// Controls the heater
//
FUNCTION_BLOCK FB_HeaterCtrl
VAR_INPUT
	
	Step: SINT; // Step counter (1...100)
	
END_VAR
VAR
	
	// Function blocks...
	fbPID: FB_CTRL_PID; // PID controller
	
	// Structures...
	stParams: ST_CTRL_PID_PARAMS; // PID controller parameters
	
	// Booleans...
	bInitialized: BOOL; // Initialized
	bRestart:     BOOL; // Restart
	bAutoStep:    BOOL; // Auto-step
	
END_VAR

// Initialize members
bRestart    := ( bRestart    OR IO_Outputs.o_Restart );

// First visit ? 
IF NOT bInitialized THEN
	
	// Initialize PID controller parameters
	bInitialized := TRUE;
	InitPidParams( ADR( stParams ));
	
	bAutoStep := FALSE;
	
END_IF

// Is the the starting step ?
IF Step = 1 THEN
  
	// Update the PID controller once per every second
	fbPID
	(
		fSetpointValue := gSetpoint,
		fActualValue   := IO_Inputs.i_HtrTemp,
		fManSyncValue  := 0,
		bSync          := FALSE,
		eMode          := SEL( bRestart, eCTRL_MODE_ACTIVE, eCTRL_MODE_RESET ),
		bHold          := FALSE,
		stParams       := stParams,
		fOut           => gPower,
		eState         => gePidState
(*
		bARWactive     => BOOL;
		eErrorId       => E_CTRL_ERRORCODES;
		bError         => BOOL;
*)
	);

	// Control the heater to ON/OFF
	IO_Outputs.o_HtrON := ( fbPID.fOut >= Step );
	bRestart           := FALSE;
	
	// Auto-step control
	IF bAutoStep THEN
		gAutoStepTimer := gAutoStepTimer+1;
		IF (gAutoStepTimer >= 20) THEN
			gSetpoint := gSetpoint + gStepChange;
			IF (gSetpoint > 200) THEN
				gSetpoint := 190;
				gStepChange := -10;
			ELSIF (gSetpoint < 0) THEN
				gSetpoint := 10;
				gStepChange := 10;
			END_IF
			gAutoStepTimer := 0;
		END_IF
	END_IF
	
// else, Not the first step now => Is heater controlled to ON ?
ELSIF IO_Outputs.o_HtrON THEN
	
	// Control the heater to ON/OFF
	IO_Outputs.o_HtrON := ( fbPID.fOut >= Step );
	
END_IF

IF IO_Outputs.o_AddTemp20 THEN
	
	gSetpoint := gSetpoint + 20;
	
	IF (gSetpoint > 200) THEN
		gSetpoint := 200;
	END_IF
	
	IO_Outputs.o_AddTemp20 :=FALSE;
	
END_IF

IF IO_Outputs.o_DropTemp20 THEN
	
	gSetpoint := gSetpoint - 20;
	
	IF (gSetpoint < 0) THEN
		gSetpoint := 0;
	END_IF
	
	IO_Outputs.o_DropTemp20 :=FALSE;
	
END_IF

IF IO_Outputs.o_AutoStep THEN
	
	IF bAutoStep THEN
		gStepChange := 10;
		gAutoStepTimer := 0;
		bAutoStep := FALSE;
		gBoolAutoStep := FALSE;
	ELSE
		bAutoStep := TRUE;
		gBoolAutoStep := TRUE;
	END_IF
	
	IO_Outputs.o_AutoStep :=FALSE;
	
END_IF

END_FUNCTION_BLOCK

(* stored: Version 1.1.0.1, ProductVersion 3.1.4022.18
   POU FB_HeaterCtrl: Id {96adc1bf-6090-4303-a06f-1b914879b476}, SpecialFunc None *)
